PROGRAM MAIN
VAR
	dummy :BOOL := FALSE;
END_VAR

//dummy := GVL.G_FromYaskawa[0].1;
//int_check();

Robot_IO_mapping();

END_PROGRAM

(* stored: Version 1.1.0.1, ProductVersion 3.1.4024.9
   POU MAIN: Id {b581cc96-544a-4433-b34c-693c6f010412}, SpecialFunc None *)
